// TwinCAT 3 PLC project main
// ProgramVersion: 3.1.4024.0
// libraries:
//   Tc2_Standard, * (Beckhoff Automation GmbH)
//   Tc2_System, * (Beckhoff Automation GmbH)
//   Tc3_Module, * (Beckhoff Automation GmbH)
// project tree:
//   / PlcTask.TcTTO
//   POUs/ MAIN.TcPOU
// real-time tasks:
//   TASK PlcTask: cycle T#10ms, priority 20, ADS port 350

CONFIGURATION main
    RESOURCE PLC ON TwinCAT3
        TASK PlcTask(INTERVAL := T#10ms, PRIORITY := 20);
        PROGRAM MAIN WITH PlcTask : MAIN;
    END_RESOURCE
END_CONFIGURATION

// ---- POUs/MAIN.TcPOU
PROGRAM MAIN
VAR
	bS1 : BOOL; //Sensor 1
	bS2 : BOOL; //Sensor 2
	bS3 : BOOL; //Sensor 3
	
	bL1 : BOOL; //Lamp 1
	bL2 : BOOL; //Lamp 2
	bL3 : BOOL; //Lamp 3
	bL4 : BOOL; //Lamp 4
	bL5 : BOOL; //Lamp 5
END_VAR

//In een vat wordt een proces bewaakt met 3 sensoren
//	* Sensor1 meet de druk. TRUE bij een te hoge druk.
//	* Sensor2 meet de temperatuur. TRUE bij een te hoge temperatuur.
//	* Sensor3 meet het vloeistofniveau. FALSE bij een te laag niveau.

//Er zijn 5 lampen die als indicator dienen voor het proces:
//	* Lamp1 gaat aan als de druk te hoog is.
//	* Lamp2 gaat aan als de temperatuur te hoog is.
//	* Lamp3 gaat aan als het niveau te laag is.
//	* Bovenstaande lampen gaan automatisch uit als er geen melding meer gegeven hoeft te worden.
//	* Lamp4 gaat aan als er zich twee alarmen gelijktijdig voordoen. Van zodra er geen twee alarmen meer zijn gaat deze lamp uit. 
//	  Bij drie alarmen gaat deze lamp ook uit.
//	* Lamp5 gaat aan als er drie alarmen zijn. Deze lamp blijft aan, ook nadat er geen drie alarmen meer zijn. 
//    De lamp kan enkel uitgeschakeld worden met een extra drukknop.

bL1 := bS1;
bL2 := bS2;
bL3 := bS3;
bL4 := (bS1 AND bS2) OR (bS1 AND bS3) OR (bS2 AND bS3) AND NOT(bS1 AND bS2 AND bS3);
bL5 :=

END_PROGRAM
